(* PLC project Unnamed, Unknown Unnamed 1 *)
(* stored: creationDateTime 2021-10-04T11:07:37, modificationDateTime 2021-10-04T13:52:55 *)

PROGRAM part4b
  VAR
    Tank1_LowLvlSensor AT %IX0.0 : BOOL;
    Tank1_MedLvlSensor AT %IX0.1 : BOOL;
    Tank1_HighLvlSensor AT %IX0.2 : BOOL;
    Tank2_LowLvlSensor AT %IX0.3 : BOOL;
    Tank2_MedLvlSensor AT %IX0.4 : BOOL;
    Tank2_HighLvlSensor AT %IX0.5 : BOOL;
    Tank3_LowLvlSensor AT %IX0.6 : BOOL;
    Tank3_MedLvlSensor AT %IX0.7 : BOOL;
    Tank3_HighLvlSensor AT %IX1.0 : BOOL;
    Tank4_LowLvlSensor AT %IX1.1 : BOOL;
    Tank4_MedLvlSensor AT %IX1.2 : BOOL;
    Tank4_HighLvlSensor AT %IX1.3 : BOOL;
    Tank1_OutValve AT %QX0.0 : BOOL;
    Tank2_OutValve AT %QX0.1 : BOOL;
    Tank3_OutValve AT %QX0.2 : BOOL;
    Tank4_OutValve AT %QX0.3 : BOOL;
  END_VAR
  VAR
    Trigger : BOOL;
    TON0 : TON;
  END_VAR

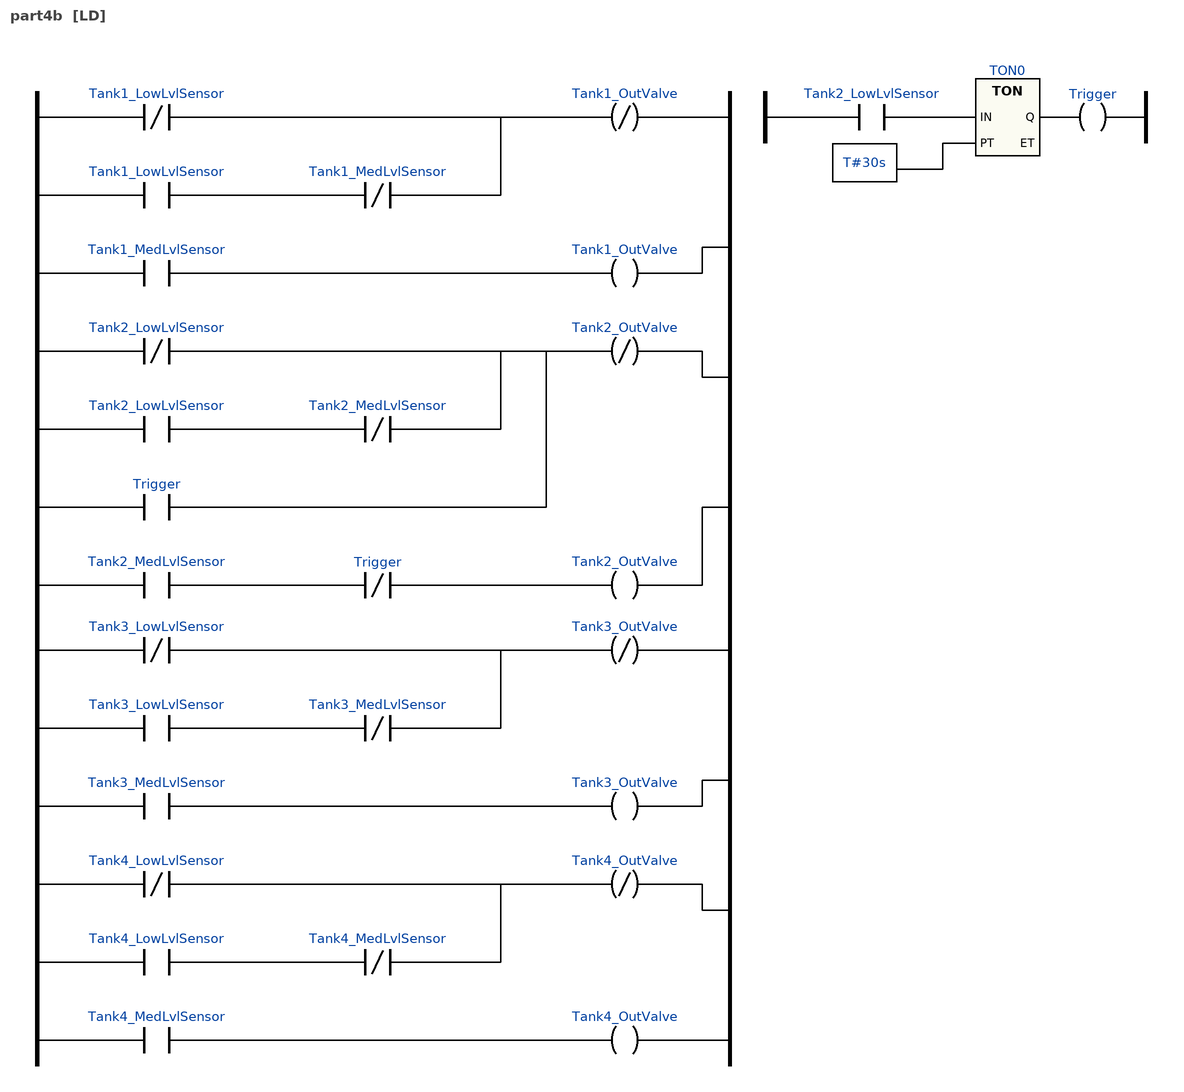
(* LD diagram, written out as Structured Text *)
Tank1_OutValve := NOT (NOT Tank1_LowLvlSensor OR Tank1_LowLvlSensor AND NOT Tank1_MedLvlSensor);
TON0(IN := Tank2_LowLvlSensor, PT := T#30s);
Trigger := TON0.Q;
Tank1_OutValve := Tank1_MedLvlSensor;
Tank2_OutValve := NOT (NOT Tank2_LowLvlSensor OR Tank2_LowLvlSensor AND NOT Tank2_MedLvlSensor OR Trigger);
Tank2_OutValve := Tank2_MedLvlSensor AND NOT Trigger;
Tank3_OutValve := NOT (NOT Tank3_LowLvlSensor OR Tank3_LowLvlSensor AND NOT Tank3_MedLvlSensor);
Tank3_OutValve := Tank3_MedLvlSensor;
Tank4_OutValve := NOT (NOT Tank4_LowLvlSensor OR Tank4_LowLvlSensor AND NOT Tank4_MedLvlSensor);
Tank4_OutValve := Tank4_MedLvlSensor;
END_PROGRAM

CONFIGURATION Config0
  RESOURCE Res0 ON PLC
    TASK task0(INTERVAL := T#20ms, PRIORITY := 0);
    PROGRAM instance0 WITH task0 : part4b;
  END_RESOURCE
END_CONFIGURATION
